// TIA Portal V16 export
// export: Created 2023-03-29T11:03:39.688751Z, ExportSetting WithDefaults, DisplayName Totally Integrated Automation Portal, DisplayVersion V16 Update 6, DisplayName TIA Portal Version Control Interface, DisplayVersion V16 Update 2, DisplayName TIA Portal Openness, DisplayVersion V16 Update 6, DisplayName STEP 7 Professional, DisplayVersion V16 Update 6, DisplayName STEP 7 Safety, DisplayVersion V16, DisplayName WinCC Advanced, DisplayVersion V16 Update 6
DATA_BLOCK "Client_ModbusTCP_sending_parameters_DB"   // DB30
AUTHOR : rtecmer
VERSION : 0.1
// stored: AutoNumber true, DBAccessibleFromOPCUA true, InstanceOfName Client_ModbusTCP_sending_parameters, InstanceOfType FB
"Client_ModbusTCP_sending_parameters"
   // VAR_IN_OUT
   //    modbustcp_przetwarzanie_in : Bool;
   //    modbustcp_przetwarzanie_out : Bool;
   // END_VAR
BEGIN
END_DATA_BLOCK
